// TIA Portal V19 export
TYPE "DiagnosticUDT"
   STRUCT
      hwID : HW_ANY;
      Count_Diag : UInt;
      RetVal : Int;
      ComponentDiag : DIS;
      SubComponentDiag : DNN;
   END_STRUCT;
END_TYPE
